PROGRAM OP130_RH_Auto
VAR
	OP130_Torque_Monitor_Dly: TON;
	OP130_Torque_Monitor_Dly_RH: TON;
	
END_VAR

CASE OP130_RH_AutoSeq OF
	10: IF (OP130_Prev_RH_COMP_OK= TRUE) AND OP130_StartEnable THEN 
		OP130_RH_AutoSeq:=20;
		END_IF
		IF (OP130_Prev_RH_COMP_NOK= TRUE) THEN 
			OP130_RH_AutoSeq:=180;
		END_IF
	
	20:IF (TRUE) AND OP130_StartEnable THEN	
		OP130_RH_AutoSeq:=30;
	   END_IF
	30:IF (OP130_GVL.SR130_RH_Servo_Control.Axis_Enabled=TRUE OR OP130_Dry_Run) AND OP130_StartEnable THEN
		OP130_RH_AutoSeq:=40;
		END_IF
	40:IF (I130_RH_ROTRY_0_DEGI1300_2=TRUE OR OP130_Dry_Run) AND OP130_StartEnable THEN
		OP130_RH_AutoSeq:=50;
		END_IF
	50:IF (OP130_StartEnable) THEN 
		OP130_GVL.SR130_RH_Vert_Servo.fTargetPosition:=OP130_GVL.SR130_HMI_LH_Servo_Work_Position;
		OP130_GVL.SR130_RH_Vert_Servo.fTargetVelocity:=OP130_GVL.SR130_HMI_LH_Servo_Work_Velocity;
		OP130_RH_AutoSeq:=60;
		END_IF
		
	60:IF(OP130_StartEnable) THEN 
		OP130_GVL.SR130_RH_Servo_Control.ABSmove_Start:=TRUE;
		OP130_RH_AutoSeq:=70;
		END_IF
	70:IF(OP130_StartEnable)AND OP130_GVL.SR130_RH_Servo_Control.Axis_In_Pos THEN 
		OP130_RH_AutoSeq:=80;
		END_IF
	80:IF (OP130_StartEnable) THEN
		  OP130_GVL.CR130_RH_Rot_Cyl.AutoCmd2:=TRUE;
		 OP130_GVL.CR130_RH_Rot_Cyl.AutoCmd1:=FALSE;
		  IF (OP130_GVL.CR130_RH_Rot_Cyl.Position2=TRUE) THEN
			  OP130_RH_AutoSeq:=90;
			  END_IF
			  
		  END_IF
	90:IF (OP130_StartEnable) THEN
		OP130_GVL.SR130_RH_Vert_Servo.fTargetPosition:=OP130_GVL.SR130_HMI_RH_Servo_Lock_Position;
		OP130_GVL.SR130_RH_Vert_Servo.fTargetVelocity:=OP130_GVL.SR130_HMI_RH_Servo_Lock_Velocity;
		  
		 OP130_RH_AutoSeq:=100;
		 END_IF
	100:IF (OP130_StartEnable) THEN
		
		OP130_GVL.SR130_RH_Servo_Control.ABSmove_Start:=TRUE;
		 OP130_RH_AutoSeq:=110;
		END_IF
    110:IF (OP130_StartEnable) AND OP130_GVL.SR130_RH_Servo_Control.Axis_In_Pos THEN
		 OP130_RH_AutoSeq:=140;
		END_IF
	
		
	140: IF (OP130_StartEnable) THEN 
          //Change TO Torque Mode
		  OP130_RH_AutoSeq:=150;
		  
		  END_IF
	
	150:IF (OP130_StartEnable) THEN
		 OP130_RH_AutoSeq:=160;  
		  END_IF
	160:IF (OP130_StartEnable) THEN
		OP130_GVL.SR130_RH_Servo_Control.ABSmove_Start:=TRUE;
		 OP130_RH_AutoSeq:=170;  
		  END_IF
	170:IF (OP130_StartEnable AND OP130_Torque_Monitor_Dly_RH.q) THEN
		IF (OP130_GVL.SR130_RH_Vert_Servo_Axis.NcToPlc.ActTorque >OP130_GVL.SR130_HMI_RH_Servo_Torque_Low_Limit) AND (OP130_GVL.SR130_RH_Vert_Servo_Axis.NcToPlc.ActTorque <SR130_HMI_RH_Servo_Torque_High_Limit) THEN
					OP130_RH_Comp_OK:=TRUE;
					OP130_RH_Comp_NOK:= FALSE;
		ELSIF(OP130_GVL.SR130_LH_Vert_Servo_Axis.NcToPlc.ActTorque <OP130_GVL.SR130_HMI_LH_Servo_Torque_Low_Limit) OR (OP130_GVL.SR130_LH_Vert_Servo_Axis.NcToPlc.ActTorque >SR130_HMI_LH_Servo_Torque_High_Limit) THEN
					OP130_RH_Comp_OK:=FALSE;
					OP130_RH_Comp_NOK:= TRUE;
					END_IF 
		IF(OP130_RH_Comp_OK OR OP130_RH_Comp_NOK) THEN
					 OP130_RH_AutoSeq:=180;	
					 END_IF
		END_IF
	
	180:IF (OP130_StartEnable) THEN
		OP130_GVL.SR130_RH_Vert_Servo.fTargetPosition:=OP130_GVL.SR130_HMI_RH_Servo_Work_Position;
		OP130_GVL.SR130_RH_Vert_Servo.fTargetVelocity:=OP130_GVL.SR130_HMI_RH_Servo_Work_Velocity;
		OP130_RH_AutoSeq:=190;
	   END_IF
	   190:IF (OP130_StartEnable) THEN
		  OP130_GVL.SR130_LH_Servo_Control.ABSmove_Start:= TRUE;
		   OP130_RH_AutoSeq:=200;
	   END_IF
	200:IF (OP130_StartEnable) AND OP130_GVL.SR130_RH_Servo_Control.Axis_In_Pos THEN
		OP130_RH_AutoSeq:=210;
	    END_IF
	210:IF  (OP130_StartEnable) THEN
		OP130_GVL.CR130_RH_Rot_Cyl.AutoCmd1:=TRUE;
		 OP130_GVL.CR130_RH_Rot_Cyl.AutoCmd2:=FALSE;
		  IF (OP130_GVL.CR130_RH_Rot_Cyl.Position1=TRUE) THEN
			  OP130_RH_AutoSeq:=220;
			  END_IF
	END_IF
	220: IF  (OP130_StartEnable) THEN
		OP130_GVL.SR130_RH_Vert_Servo.fTargetPosition:=SR130_RH_Servo_Home_Position;
		OP130_GVL.SR130_RH_Vert_Servo.fTargetVelocity:=SR130_RH_Servo_Home_Velocity;
		 OP130_RH_AutoSeq:=230;
	END_IF
	230: IF (OP130_StartEnable) THEN 
		OP130_GVL.SR130_RH_Servo_Control.ABSmove_Start:= TRUE ;
		 OP130_RH_AutoSeq:=240;
	END_IF
	
	240: IF (OP130_StartEnable) AND OP130_GVL.SR130_RH_Servo_Control.Axis_In_Pos THEN 
		 OP130_RH_AutoSeq:=250;
	END_IF
	 250:IF (OP130_StartEnable) THEN
		 OP130_RH_Operation_Completed:= TRUE;
		  OP130_RH_AutoSeq:=260;
	 END_IF

	   
END_CASE
//Torque Monitor Dly
 OP130_Torque_Monitor_Dly_RH(IN:=OP130_RH_AutoSeq=170 , PT:=T#200MS , Q=> , ET=> );

END_PROGRAM

(* stored: Version 1.1.0.1, ProductVersion 3.1.4024.11
   POU OP130_RH_Auto: Id {5e73add9-8522-4abf-9c2d-6575bca741fe}, SpecialFunc None *)
